FUNCTION_BLOCK Wago636 (* Wago 750-636 DC-Drive-Controller 24V 5A *)
  (* Standard: 61499-2; Description: Copyright (c) 2025 Monika Wenger This program and the accompanying materials are made available under the terms of the Eclipse Public License 2.0 which is available at https://www.eclipse.org/legal/epl-2.0/ SPDX-License-Identifier: EPL-2.0 *)
  (* Version 3.0, 2026-07-20, Monika Wenger, change package *)
  (* Version 1.0, 2025-05-05, Monika Wenger *)
  PACKAGE eclipse4diac::io::wago;
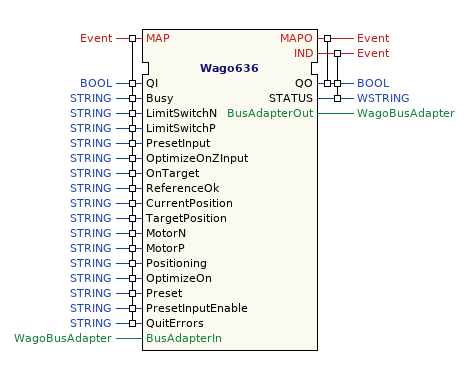
  EVENT_INPUT
    MAP WITH LimitSwitchP, LimitSwitchN, QI, MotorP, MotorN, CurrentPosition, TargetPosition, QuitErrors, Positioning, Preset, Busy, OptimizeOnZInput, OnTarget, ReferenceOk, OptimizeOn, PresetInput, PresetInputEnable; (* Map Pins *)
  END_EVENT
  EVENT_OUTPUT
    MAPO WITH QO; (* Confirm Pin Mapping *)
    IND WITH QO, STATUS; (* Indication from Resource *)
  END_EVENT
  VAR_INPUT
    QI : BOOL; (* Event Input Qualifier *)
    Busy : STRING; (* True as long as command is executed as IX *)
    LimitSwitchN : STRING; (* Reference switch negative (Hardware pin) as IX *)
    LimitSwitchP : STRING; (* Reference switch positive (Hardware Pin) as IX *)
    PresetInput : STRING; (* (Hardware pin) IX *)
    OptimizeOnZInput : STRING; (* (Hardware pin) IX *)
    OnTarget : STRING; (* True when Positioning ended at target area as IX *)
    ReferenceOk : STRING; (* True when reference movement was successfull as IX *)
    CurrentPosition : STRING; (* Current position as ID *)
    TargetPosition : STRING; (* Target position as QD *)
    MotorN : STRING; (* Motor A- (Hardware pin) as QX *)
    MotorP : STRING; (* Motor A+ (Hardware pin) as QX *)
    Positioning : STRING; (* Drive to target position (MotorN, MotorP = false) as QX *)
    OptimizeOn : STRING; (* turn prestop optimization on as QX *)
    Preset : STRING; (* A rising edge copies the target position into the current position as QX *)
    PresetInputEnable : STRING; (* preset input enabled (OptimizeOnZInput means optimize on), preset input disbaled (OptimizeOnZInput means z input) as QX *)
    QuitErrors : STRING; (* Quits error Bits as QX *)
  END_VAR
  VAR_OUTPUT
    QO : BOOL; (* Event Output Qualifier *)
    STATUS : WSTRING; (* Service Status *)
  END_VAR
  SOCKETS
    BusAdapterIn : eclipse4diac::io::wago::WagoBusAdapter;
  END_SOCKETS
  PLUGS
    BusAdapterOut : eclipse4diac::io::wago::WagoBusAdapter;
  END_PLUGS
END_FUNCTION_BLOCK
